// TIA Portal V21 export
DATA_BLOCK "HMI_Counters_DB"   // DB701
{ S7_Optimized_Access := 'TRUE' }
// stored: AutoNumber false, DBAccessibleFromWebserver false, MemoryReserve 100
   VAR
      ResetCounters { ExternalAccessible := 'False'; ExternalVisible := 'False'; ExternalWritable := 'False'} : Bool;
   END_VAR
   VAR RETAIN
      Machine : "UDT_WORK_CNT";
      Pump : Array[1..2] of "UDT_WORK_CNT";
   END_VAR
BEGIN
END_DATA_BLOCK
